RoboDK station: RDTSDemoBasketLine.rdk

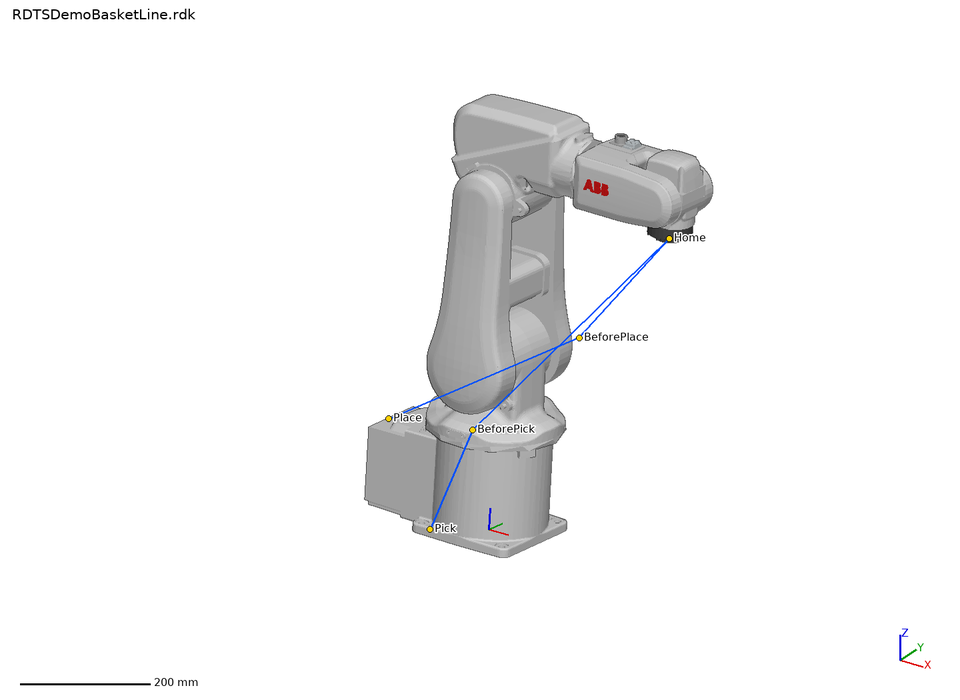
[picture v0: the station drawn from its stored meshes, robots at their saved joint values, targets as dots, program paths as lines]
Station RDTSDemoBasketLine (saved by RoboDK 5.6.0). Poses are relative to the parent item; angles as X-Y-Z fixed-axis rotations.
Station parameters (name, value as stored): 1MoveToPick, 0, 1MakePick, 0, 1PickObjOK, 0, 1MoveToPlace, 0, 1MakePlace, 0, 1PlaceObjOK, 0, 1Waitting, 1, 2MoveToPick, 0, 2MakePick, 0, 2PickObjOK, 0, 2MoveToPlace, 0, 2MakePlace, 0, 2PlaceObjOK, 0, 2Waitting, 1, 3MoveToPick, 0, 3MakePick, 0, 3PickObjOK, 0, 3MoveToPlace, 0, 3MakePlace, 0, 3PlaceObjOK, 0, 3Waitting, 1, 4MoveToPick, 0, 4MakePick, 0, 4PickObjOK, 0, 4MoveToPlace, 0, 4MakePlace, 0, 4PlaceObjOK, 0, 4Waitting, 1
  - frame Robot1Base at (0, 0, 0) mm, rotated rx -6.07 ry -0.54 rz 0 deg
    - robot Robot1 (model ABB IRB 120-3/0.6): 6 axes, payload 3 kg, reach 580 mm, repeatability 0.01 mm, weight 25 kg
        modified DH rows (alpha deg, a mm, theta deg, d mm): 0, 0, 0, 290; -90, 0, -90, 0; 0, 270, 0, 0; -90, 70, 0, 302; 90, 0, 0, 0; -90, 0, 180, 72
        joint limits [-165, -110, -90, -160, -120, -400] to [165, 110, 70, 160, 120, 400]; home [0, 0, 0, 0, 0, 0]; saved at [0, 0, 0, 0, 90, 0]
    - target Home (Cartesian target) at (302, 0, 558) mm, rotated rx 180 ry 0 rz -180 deg; joints [0, 0, 0, 0, 90, 0] of Robot1
    - target BeforePick (Cartesian target) at (172.08, -318.94, 298.42) mm, rotated rx -82.15 ry -59.79 rz 80.08 deg; joints [-52.941, 39.526, 14.87, -57.623, 115.507, 0.453] of Robot1
    - target Pick (Cartesian target) at (159.34, -401.71, 154.17) mm, rotated rx -82.15 ry -59.79 rz 80.08 deg; joints [-60.332, 71.35, -11.192, -62.618, 109.176, 3.69] of Robot1
    - target AfterPick (Cartesian target) at (172.08, -318.94, 298.42) mm, rotated rx -82.15 ry -59.79 rz 80.08 deg; joints [-52.941, 39.526, 14.87, -57.623, 115.507, 0.453] of Robot1
    - target BeforePlace (Cartesian target) at (302, -233.4, 459.61) mm, rotated rx 180 ry 0 rz 180 deg; joints [-37.699, 15.517, 0.964, 0, 73.519, -37.699] of Robot1
    - target BeforePlace2 (Cartesian target) at (302, -233.4, 459.61) mm, rotated rx 180 ry 0 rz 180 deg; joints [-37.699, 15.517, 0.964, 0, 73.519, -37.699] of Robot1
    - target Place (Cartesian target) at (18.87, -323.47, 277.74) mm, rotated rx -152.18 ry 18.03 rz 149.61 deg; joints [-86.206, 13.153, 43.71, -77.787, 2.099, 25.863] of Robot1
    - target AfterPlace (Cartesian target) at (302, -233.4, 459.61) mm, rotated rx 180 ry 0 rz 180 deg; joints [-37.699, 15.517, 0.964, 0, 73.519, -37.699] of Robot1
    - target AfterPlace2 (Cartesian target) at (302, -233.4, 459.61) mm, rotated rx 180 ry 0 rz 180 deg; joints [-37.699, 15.517, 0.964, 0, 73.519, -37.699] of Robot1
  - program RobotProg1 (30 instructions, listed below)
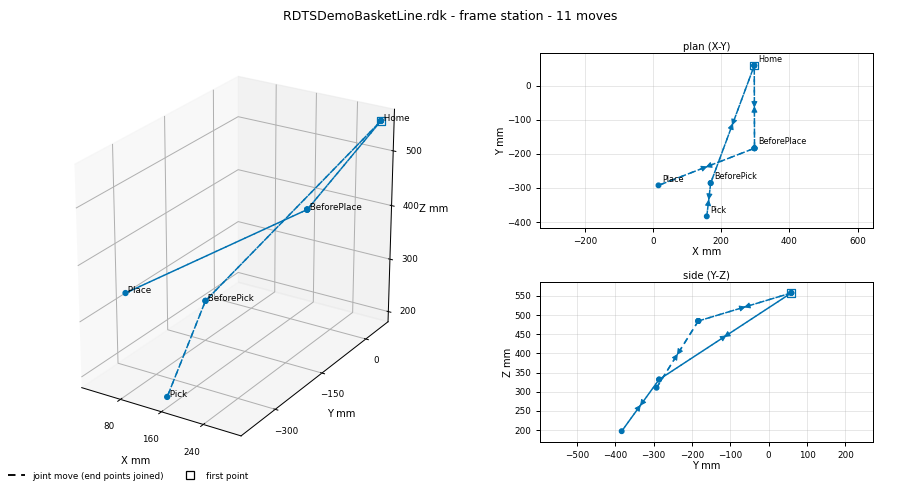
[picture p0: tool path of RDTSDemoBasketLine.rdk in frame station, 11 of 11 moves have a stored position in this frame; points joined in program order, loops and branches not executed]

--- program RobotProg1 (robot Robot1) ---
  设置参考: Robot1Base
  MoveJ (Home)
  Set 1MakePick=0
  Set 1PickObjOK=0
  Set 1MakePlace=0
  Set 1PlaceObjOK=0
  Wait 1MoveToPick=1
  Set 1Waitting=0
  MoveJ (BeforePick)
  MoveJ (Pick)
  Set 1MakePick=1
  Wait 1PickObjOK=1
  Set 1MakePick=0
  暂停 2.0 s
  MoveJ (AfterPick)
  MoveJ (Home)
  Set 1Waitting=1
  Wait 1MoveToPlace=1
  Set 1Waitting=0
  MoveJ (BeforePlace)
  MoveJ (BeforePlace2)
  MoveJ (Place)
  Set 1MakePlace=1
  Wait 1PlaceObjOK=1
  Set 1MakePlace=0
  暂停 1.0 s
  MoveJ (AfterPlace)
  MoveJ (AfterPlace2)
  MoveJ (Home)
  Set 1Waitting=1
